_CFC_ (* Continuous Function Chart, elements in execution order *)
#0 fb_HVACAO_SCHU_P2_1_YA3_AO3:FB_HVACAnalogOutput(eHVACDataSecurityType_Idle, FALSE, TRUE, SCHU_P2_1_YA3_ZAD_VN, TRUE, eHVACAnalogOutputMode_Auto_BMS, -, -, -, SCHU_P2_1_SB, YA_HIGHRANGE, YA_LOWRANGE, direction, enableFeedbCtrl, hysFbCtrl, delay)
#1 SCHU_P2_1_YA3_AO3 <= #0.out 2
#2 OR(#0.out 7, #0.out 9)
#3 YA3_AO_OTKAZ <= #2
_END_CFC_
END_PROGRAM

(* POU Output/AO/YA4_Z, CFC *)
PROGRAM YA4_Z
VAR
	fb_HVACAO_SCHU_P2_1_YA4_AO4: FB_HVACAnalogOutput;
	enableFeedbCtrl: BOOL := FALSE;
	hysFbCtrl: REAL := 0;
	direction: BOOL;
	delay: TIME := T#0s;
END_VAR
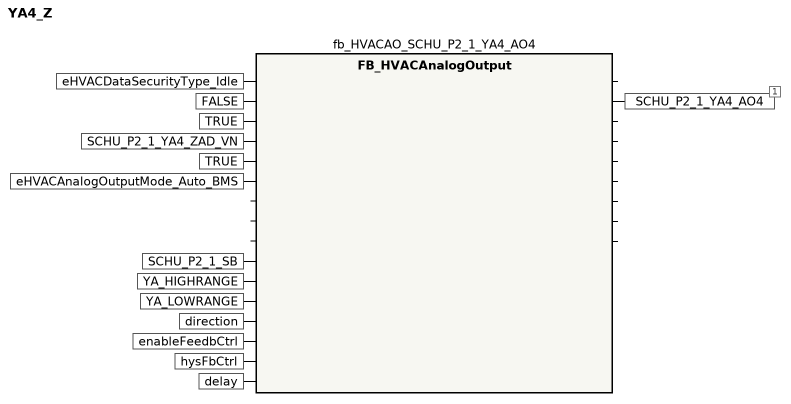
_CFC_ (* Continuous Function Chart, elements in execution order *)
#0 fb_HVACAO_SCHU_P2_1_YA4_AO4:FB_HVACAnalogOutput(eHVACDataSecurityType_Idle, FALSE, TRUE, SCHU_P2_1_YA4_ZAD_VN, TRUE, eHVACAnalogOutputMode_Auto_BMS, -, -, -, SCHU_P2_1_SB, YA_HIGHRANGE, YA_LOWRANGE, direction, enableFeedbCtrl, hysFbCtrl, delay)
#1 SCHU_P2_1_YA4_AO4 <= #0.out 2
_END_CFC_
END_PROGRAM

(* POU Input/ModBus/MB_UZT, CFC *)
PROGRAM MB_UZT
VAR
	MB_READ_REGS: ModbusRtuMaster_KL6x22B;
	Quantity: WORD:= 4;
	MBAddr: WORD:= 16#3000;
	Error: BOOL;
	Errorld: MODBUS_ERRORS;
	cbRead: UINT;

	TON1: TON;

	UnitID_2: BYTE:=2;
	rs_s: RS;
	UnitID_1: BYTE := 1;

	SWT: BOOL;
	ton2: TON;
	tp1: TOF;

END_VAR
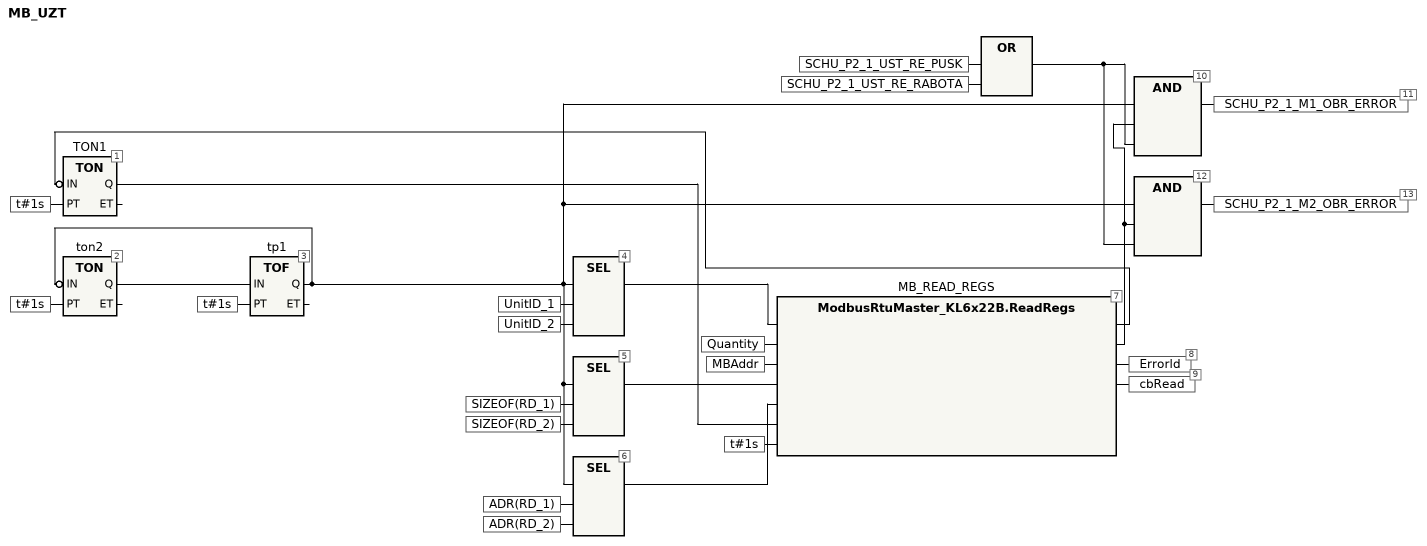
_CFC_ (* Continuous Function Chart, elements in execution order *)
#0 OR(SCHU_P2_1_UST_RE_PUSK, SCHU_P2_1_UST_RE_RABOTA)
#1 TON1:TON(IN: NOT #7.out 1, PT: t#1s)
#2 ton2:TON(IN: NOT #3.Q, PT: t#1s)
#3 tp1:TOF(IN: #2.Q, PT: t#1s)
#4 SEL(#3.Q, UnitID_1, UnitID_2)
#5 SEL(#3.Q, SIZEOF(RD_1), SIZEOF(RD_2))
#6 SEL(#3.Q, ADR(RD_1), ADR(RD_2))
#7 MB_READ_REGS:ModbusRtuMaster_KL6x22B.ReadRegs(#4, Quantity, MBAddr, #5, #6, #1.Q, t#1s)
#8 Errorld <= #7.out 3
#9 cbRead <= #7.out 4
#10 AND(#3.Q, #7.out 2, #0)
#11 SCHU_P2_1_M1_OBR_ERROR <= #10
#12 AND(#3.Q, #7.out 2, #0)
#13 SCHU_P2_1_M2_OBR_ERROR <= #12
_END_CFC_
END_PROGRAM
